TYPE ZDataRecipe :
STRUCT
  RecipeParam1 : LREAL;
  RecipeParam2 : LREAL;
  RecipeParam3 : LREAL;
END_STRUCT
END_TYPE

(* stored: Version 1.1.0.1
   DUT ZDataRecipe: Id {940adc8c-1eee-4505-b23a-b0b20f8a18c6} *)
